Fanuc KAREL source: compact_preamble.KL

PROGRAM KT00372
%NOLOCKGROUP
VAR
R1:REAL
H2 : ARRAY[2] OF SHORT
OUT:BOOLEAN
BEGIN
R1=2.0
H2[1]=3
OUT=(R1 <=(H2[1]))
END KT00372
